FUNCTION_BLOCK GripperSkill (* Basic FB with empty ECC *)
  (* Standard: 61499-2 *)
  (* Version 1.0, 2021-09-15, dorofeev *)
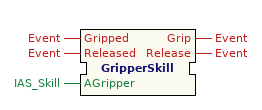
  EVENT_INPUT
    Gripped;
    Released;
  END_EVENT
  EVENT_OUTPUT
    Grip;
    Release;
  END_EVENT
  SOCKETS
    AGripper : IAS_Skill;
  END_SOCKETS
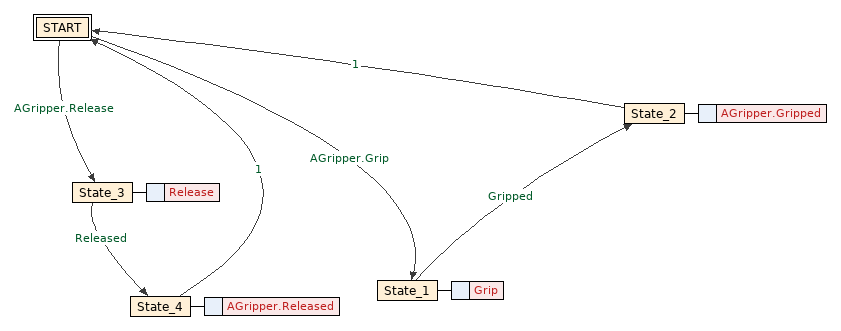
  EC_STATES
    START; (* Initial State *)
    State_1 : -> Grip;
    State_2 : -> AGripper.Gripped;
    State_3 : -> Release;
    State_4 : -> AGripper.Released;
  END_STATES
  EC_TRANSITIONS
    State_1 TO State_2 := Gripped;
    State_3 TO State_4 := Released;
    START TO State_3 := AGripper.Release;
    State_4 TO START := 1;
    START TO State_1 := AGripper.Grip;
    State_2 TO START := 1;
  END_TRANSITIONS
END_FUNCTION_BLOCK
